FUNCTION_BLOCK FB_PulseTrainControl
VAR_INPUT
END_VAR
VAR_OUTPUT
END_VAR
VAR
	pPulseTrainChannel : POINTER TO ST_PulseTrainChannel;
	nFrequency : UINT;
END_VAR

METHOD M_GetFrequency : UINT
VAR_INPUT
END_VAR
M_GetFrequency := nFrequency;
END_METHOD

METHOD M_GetPulse : UINT
VAR_INPUT
END_VAR
IF pPulseTrainChannel > 0 THEN
	M_GetPulse := pPulseTrainChannel^.nPulse;
END_IF
END_METHOD

METHOD M_SetFrequency : ERRORID
VAR_INPUT
	nValue : UINT;
END_VAR
IF pPulseTrainChannel = 0 THEN
	M_SetFrequency := E_ErrorIdObjMgmt.ERRORID_InvalidTriggerChannel;
	RETURN;
END_IF
IF nValue >= 16 AND nValue <= 10000 THEN
	nFrequency := nValue;
	pPulseTrainChannel^.nPeriod := UDINT_TO_UINT(1000000 / nFrequency);
ELSE
	M_SetFrequency := E_ErrorIdObjMgmt.ERRORID_InvalidFrequency;
END_IF
END_METHOD

METHOD M_SetPulse : ERRORID
VAR_INPUT
	nValue : UINT;
END_VAR
IF pPulseTrainChannel = 0 THEN
	M_SetPulse := E_ErrorIdObjMgmt.ERRORID_InvalidTriggerChannel;
	RETURN;
END_IF
IF nValue > 0 AND nValue <= 65635 THEN
	pPulseTrainChannel^.nPulse := nValue;
ELSE
	M_SetPulse := E_ErrorIdObjMgmt.ERRORID_InvalidPulseWidth;
END_IF
END_METHOD

METHOD M_SetPulseTrainChannel
VAR_INPUT
	pPulseTrainChannel : POINTER TO ST_PulseTrainChannel;
END_VAR
THIS^.pPulseTrainChannel := pPulseTrainChannel;
END_METHOD

METHOD M_Start
VAR_INPUT
	nNrOfPulses : UINT;
END_VAR
IF pPulseTrainChannel > 0 THEN
	pPulseTrainChannel^.nNoOfPulses := nNrOfPulses;
	pPulseTrainChannel^.nCtrl := 1;
END_IF
END_METHOD

METHOD M_Stop
VAR_INPUT
END_VAR
IF pPulseTrainChannel > 0 THEN
	pPulseTrainChannel^.nCtrl := 0;
END_IF
END_METHOD

PROPERTY P_bBusy : BOOL
GET
IF pPulseTrainChannel > 0 THEN
	P_bBusy := pPulseTrainChannel^.nState.0;
END_IF
END_GET
END_PROPERTY

END_FUNCTION_BLOCK

(* stored: Version 1.1.0.1, ProductVersion 3.1.4022.12
   POU FB_PulseTrainControl: Id {4e94401d-c1c7-48b6-af12-c6dac1216317}, SpecialFunc None
   Method M_GetFrequency: Id {7d5645c0-644c-4d57-a080-a85fdc85682e}
   Method M_GetPulse: Id {ef55df2c-cf1a-427f-b88f-348ce810c547}
   Method M_SetFrequency: Id {85334777-6d9e-43b4-b823-c238eb39883f}
   Method M_SetPulse: Id {3a21dcf7-c0ad-4c98-a25c-aa22cd473a78}
   Method M_SetPulseTrainChannel: Id {d57af17d-521b-4ad9-899d-0bd58d71e661}
   Method M_Start: Id {345143db-58b2-429d-a443-c788f0a8c2b7}
   Method M_Stop: Id {cb9ad9e6-dac3-43cc-97e2-ef84f8607eb5}
   Property P_bBusy: Id {13d633f0-2cfa-49bd-89fc-a3183b13522a}
   Get Get: Id {e8acd363-c099-4731-adfe-9c0d7d80a410} *)
